{attribute 'monitoring' := 'call'}
PROPERTY OID : CHALET_BaseComponents.OTCID
GET
END_GET
END_PROPERTY

END_INTERFACE

// COMPONENTs/VnRegister-Access/FB_VnRegister_UDINT
{attribute 'no_explicit_call' := 'Do not call the body - Stick to OOP'}
FUNCTION_BLOCK FB_VnRegister_UDINT EXTENDS FB_VnRegister_Base
VAR
	{attribute 'hide'}
	nValue : UDINT;
	
	{attribute 'hide'}	
	fbVnReadRegister_UDINT : FB_VN_ReadRegister_UDINT;
	{attribute 'hide'}
	fbVnWriteRegister_UDINT : FB_VN_WriteRegister_UDINT;
END_VAR

METHOD FB_init : BOOL
VAR_INPUT
	bInitRetains : BOOL; // if TRUE, the retain variables are initialized (warm start / cold start)
	bInCopyCode : BOOL;  // if TRUE, the instance afterwards gets moved into the copy code (online change)
	
	ipCameraConnection : I_GigEVision_Register_Connection;
	nAddress : GVCP_REGISTER_ADDRESS;
    nEndian  : UINT;
END_VAR
VAR_INST
	{attribute 'hide'}
	bFBInitCalledOnce : BOOL; //Do the following code once during start up and not during onlinechange
END_VAR
//Do the following code once during start up and not during onlinechange
IF NOT bFBInitCalledOnce THEN 
	nCtsVnRegisterObject := nCtsVnRegisterObject +1;
	

	THIS^.nEndian 		:= nEndian;
	
	//Copy ObjectId from Camera to this fbVnReadRegister.
	MEMCPY(destAddr := ADR(fbVnReadRegister_UDINT.oidITcVnGevImageProvider), srcAddr:=ADR(SUPER^.OidCamera), n:= SIZEOF(SUPER^.OidCamera));
	MEMCPY(destAddr := ADR(fbVnWriteRegister_UDINT.oidITcVnGevImageProvider), srcAddr:=ADR(SUPER^.OidCamera), n:= SIZEOF(SUPER^.OidCamera));

	//Force to do an init after set OID
	fbVnReadRegister_UDINT.FB_init(FALSE,FALSE);	
	fbVnWriteRegister_UDINT.FB_init(FALSE,FALSE);
END_IF

bFBInitCalledOnce := TRUE;
END_METHOD

METHOD Update : HRESULT
SUPER^.Update();


fbVnReadRegister_UDINT(
	nAddress:= SUPER^.nAddress, 
	nEndian:= SUPER^.nEndian, 
	bRead:= SUPER^.bExecuteRead, 
	bBusy=> SUPER^.bReadBusy, 
	bError=> SUPER^.bReadError
	);
IF fbRTrigReadDone.Q AND THIS^.bWriteDone THEN
	nValue := fbVnReadRegister_UDINT.nValue;
END_IF
	
	
fbVnWriteRegister_UDINT(
	nAddress:= SUPER^.nAddress, 
	nValue:= nValue,  
	nEndian:= SUPER^.nEndian,   
	bWrite:= SUPER^.bExecuteWrite, 
	bBusy=> SUPER^.bWriteBusy, 
	bError=> SUPER^.bWriteError,
	);
END_METHOD

{attribute 'monitoring':='call'}
PROPERTY Value : UDINT
GET
Value := nValue;
END_GET
SET
nValue := Value;

//Trigger a new write cycle
THIS^.bWriteDone 	:= FALSE;
END_SET
END_PROPERTY

END_FUNCTION_BLOCK

// COMPONENTs/VnRegister-Access/internal/FB_VnRegister_Base
(* This FB is abstract and is the base class  *)
FUNCTION_BLOCK ABSTRACT FB_VnRegister_Base EXTENDS FB_CH_Object IMPLEMENTS I_VnRegister_Status
VAR

	{attribute 'hide'}
	bErrorInvalideInterface : BOOL;
	
	{attribute 'hide'}	
	OidCamera : OTCID;
	{attribute 'hide'}
	//The address of the first byte to write to the camera 
    nAddress : GVCP_REGISTER_ADDRESS;
	{attribute 'hide'}
	//The endianness of the register. 0 = Big, 1 = Little. Default: 0
    nEndian  : UINT;
	
	//in the event of a connection interruption to the device, either a read under write command is repeated
	{attribute 'hide'}
	eCommandToRepeadAfterReconnect : (READ, WRITE) := READ;
	
	//Read/write 
	{attribute 'hide'}
	bReadDone : BOOL;
	{attribute 'hide'}
	fbRTrigReadDone : R_TRIG();
	{attribute 'hide'}
	nSeqRead : UINT;
	{attribute 'hide'}
	bExecuteRead : BOOL;
	{attribute 'hide'}
	bReadError : BOOL;
	{attribute 'hide'}
	bReadBusy : BOOL;
	
	{attribute 'hide'}
	bWriteDone : BOOL := TRUE;
	{attribute 'hide'}
	nSeqWrite : UINT;

	{attribute 'hide'}
	bExecuteWrite : BOOL;	
	{attribute 'hide'}
	bWriteError : BOOL;
	{attribute 'hide'}
	bWriteBusy : BOOL;
	
	{attribute 'hide'}
	fbDelayOnError : TON := ( PT:= T#100MS);
END_VAR
VAR_STAT
	{attribute 'hide'}
	nCtsVnRegisterObject : UDINT;
	{attribute 'hide'}
	nCtsReadActive : UDINT;
	{attribute 'hide'}
	nCtsWriteActive : UDINT;
END_VAR

{attribute 'monitoring':='call'}
PROPERTY Error : BOOL
GET
Error := THIS^.bReadError OR THIS^.bWriteError OR THIS^.bErrorInvalideInterface;
END_GET
END_PROPERTY

METHOD FB_init : BOOL
VAR_INPUT
	bInitRetains : BOOL; // if TRUE, the retain variables are initialized (warm start / cold start)
	bInCopyCode : BOOL;  // if TRUE, the instance afterwards gets moved into the copy code (online change)
	
	ipCameraConnection : I_GigEVision_Register_Connection;
    nAddress : GVCP_REGISTER_ADDRESS;
END_VAR

VAR_INST
	{attribute 'hide'}
	bFBInitCalledOnce : BOOL; //Do the following code once during start up and not during onlinechange
END_VAR
//Do the following code once during start up and not during onlinechange
IF NOT bFBInitCalledOnce THEN 
	THIS^.nAddress 		:= nAddress;

	IF ipCameraConnection <> 0 THEN
		OidCamera := ipCameraConnection.OID;
	ELSE
		bErrorInvalideInterface := TRUE;
	END_IF
END_IF

bFBInitCalledOnce := TRUE;
END_METHOD

METHOD Initialize : HRESULT
IF eCommandToRepeadAfterReconnect = READ THEN
	//the reading of the parameter should be restarted again
	THIS^.bReadDone := FALSE;
END_IF

IF eCommandToRepeadAfterReconnect = WRITE THEN
	//the reading of the parameter should be restarted again
	THIS^.bWriteDone := FALSE;
END_IF


Initialize := S_OK;
END_METHOD

{attribute 'monitoring':='call'}
PROPERTY OID : OTCID
GET
OID := OidCamera;
END_GET
END_PROPERTY

{attribute 'monitoring':='call'}
PROPERTY ReadDone : BOOL
GET
ReadDone := bReadDone;
END_GET
SET
//Only allow set to FALSE
IF NOT ReadDone THEN
	bReadDone := FALSE;
END_IF
END_SET
END_PROPERTY

METHOD Update : HRESULT
IF bErrorInvalideInterface THEN
	//Error
	RETURN;
END_IF


(*--- Read ---*)
bExecuteRead := FALSE;
CASE nSeqRead OF
	0: //Start/Restart if required
		IF NOT bReadDone  AND bWriteDone(* Write has higher priority*) AND (nCtsReadActive < VisionParameterlist.MAX_VN_REGISTER_READ) AND (nSeqWrite = 0) THEN
			bExecuteRead := TRUE; // Rising edge	
			nCtsReadActive := nCtsReadActive +1;	
			nSeqRead := 1;
		END_IF
	
	1: //Check if done or error
		IF bReadError THEN
			//Error
			nSeqRead := 99;
			fbDelayOnError.IN := TRUE;
			nCtsReadActive := nCtsReadActive -1;	
			
		ELSIF NOT bReadBusy AND NOT bReadError THEN
			//Done
			THIS^.bReadDone := TRUE;
			nSeqRead := 0;
			nCtsReadActive := nCtsReadActive -1;	
			
		ELSE
			;//Busy
		END_IF	
		
	99: // Delay on error to reduce amount of errors
		IF fbDelayOnError.Q THEN
			fbDelayOnError.IN := FALSE;
			nSeqRead := 0;
		END_IF
END_CASE

fbRTrigReadDone(CLK := THIS^.bReadDone);




(*--- Write ---*)
bExecuteWrite := FALSE;
CASE nSeqWrite OF
	0: //Start/Restart if required
		IF NOT bWriteDone AND (nCtsWriteActive < VisionParameterlist.MAX_VN_REGISTER_WRITE) AND (nSeqRead = 0) THEN
			bExecuteWrite := TRUE; // Rising edge	
			nCtsWriteActive := nCtsWriteActive +1;	
			nSeqWrite := 1;
		END_IF
	
	1: //Check if done or error
		IF bWriteError THEN
			//Error
			nSeqWrite := 99;
			fbDelayOnError.IN := TRUE;
			nCtsWriteActive := nCtsWriteActive -1;	
			
		ELSIF NOT bWriteBusy AND NOT bWriteError THEN
			//Done
			THIS^.bWriteDone := TRUE;
			nSeqWrite := 0;
			nCtsWriteActive := nCtsWriteActive -1;
			
		ELSE
			;//Busy
		END_IF	
		
	99: // Delay on error to reduce amount of errors
		IF fbDelayOnError.Q THEN
			fbDelayOnError.IN := FALSE;
			nSeqWrite := 0;
		END_IF		

END_CASE



//Update
fbDelayOnError();
END_METHOD

{attribute 'monitoring':='call'}
PROPERTY WriteDone : BOOL
GET
WriteDone := bWriteDone;
END_GET
SET
//Only allow set to FALSE
IF NOT WriteDone THEN
	bWriteDone := FALSE;
END_IF

//in the event of a connection interruption to the device, either a read under write command is repeated
eCommandToRepeadAfterReconnect := WRITE;
END_SET
END_PROPERTY

END_FUNCTION_BLOCK

// COMPONENTs/VnRegister-Access/internal/I_VnRegister_Status
INTERFACE I_VnRegister_Status

{attribute 'monitoring':='call'}
PROPERTY ReadDone : BOOL
GET
END_GET
END_PROPERTY

{attribute 'monitoring':='call'}
PROPERTY WriteDone : BOOL
GET
END_GET
END_PROPERTY

END_INTERFACE

// COMPONENTs/VnRegister-Access/FB_VnRegister_Memory
{attribute 'no_explicit_call' := 'Do not call the body - Stick to OOP'}
FUNCTION_BLOCK FB_VnRegister_Memory EXTENDS FB_VnRegister_Base
VAR
	{attribute 'hide'}
	ValueBuffer 			: ARRAY[0..535] OF BYTE;
	nLength       : UINT;
	
	{attribute 'hide'}	
	fbVnReadRegister_Memory	: FB_VN_ReadMemory;
	{attribute 'hide'}
	fbVnWriteRegister_Memory : FB_VN_WriteMemory;
END_VAR

METHOD FB_init : BOOL
VAR_INPUT
	bInitRetains : BOOL; // if TRUE, the retain variables are initialized (warm start / cold start)
	bInCopyCode : BOOL;  // if TRUE, the instance afterwards gets moved into the copy code (online change)
	
	ipCameraConnection : I_GigEVision_Register_Connection;
	nAddress : GVCP_REGISTER_ADDRESS;
	//The number of bytes to write, starting at nAddress (must be a multiple of 4, not more than 536)
	nLength       : UINT; 
END_VAR
VAR_INST
	{attribute 'hide'}
	bFBInitCalledOnce : BOOL; //Do the following code once during start up and not during onlinechange
END_VAR
//Do the following code once during start up and not during onlinechange
IF NOT bFBInitCalledOnce THEN 
	nCtsVnRegisterObject := nCtsVnRegisterObject +1;
	

	THIS^.nLength 		:=  LIMIT(4, nLength, 536);
	
	//Copy ObjectId from Camera to this fbVnReadRegister.
	MEMCPY(destAddr := ADR(fbVnReadRegister_Memory.oidITcVnGevImageProvider), srcAddr:=ADR(SUPER^.OidCamera), n:= SIZEOF(SUPER^.OidCamera));
	MEMCPY(destAddr := ADR(fbVnWriteRegister_Memory.oidITcVnGevImageProvider), srcAddr:=ADR(SUPER^.OidCamera), n:= SIZEOF(SUPER^.OidCamera));

	//Force to do an init after set OID
	fbVnReadRegister_Memory.FB_init(FALSE,FALSE);	
	fbVnWriteRegister_Memory.FB_init(FALSE,FALSE);
END_IF

bFBInitCalledOnce := TRUE;
END_METHOD

METHOD ReadData : BOOL
VAR_INPUT
	//ADR(destination)
	pBuffer  : PVOID; 
END_VAR
MEMCPY(destAddr := pBuffer, srcAddr:=ADR(ValueBuffer), n:= nLength);
END_METHOD

METHOD Update : HRESULT
SUPER^.Update();

fbVnReadRegister_Memory(
	nAddress:= SUPER^.nAddress, 
	nLength:= nLength, 
	pBuffer:= ADR(ValueBuffer), 
	bRead:= SUPER^.bExecuteRead, 
	bBusy=> SUPER^.bReadBusy, 
	bError=> SUPER^.bReadError
	);
	
fbVnWriteRegister_Memory(
	nAddress:= SUPER^.nAddress, 
	nLength:= nLength, 
	pData:= ADR(ValueBuffer), 
	bWrite:= SUPER^.bExecuteWrite, 
	bBusy=> SUPER^.bWriteBusy, 
	bError=> SUPER^.bWriteError,
	);
END_METHOD

METHOD WriteData : BOOL
VAR_INPUT
	//ADR(source)
	pBuffer  : PVOID; 
END_VAR
MEMCPY(destAddr := ADR(ValueBuffer), srcAddr:= pBuffer, n:= nLength);

//Trigger a new write cycle
THIS^.bWriteDone 	:= FALSE;
END_METHOD

END_FUNCTION_BLOCK

// COMPONENTs/ImageProvider/Camera/FB_GigE_Vision
{attribute 'no_explicit_call' := 'Do not call the body - Stick to OOP'}
FUNCTION_BLOCK FB_GigE_Vision EXTENDS FB_ImageProvider_Base IMPLEMENTS I_GigEVision_Mode, I_GigEVision_Register_Connection
VAR
	fbCamera 						: FB_VN_GevCameraControl;	// Interface object for camera use
	
	{attribute 'hide'}
	fbCameraWriteExposureTime		: FB_VN_WriteRegister_UDINT;// Interface object for camera configuration
	{attribute 'hide'}
	bResetCommand	: BOOL;
END_VAR

{attribute 'monitoring' := 'call'}
PROPERTY Exposure_1us : UDINT
GET
Exposure_1us := THIS^.fbCameraWriteExposureTime.nValue;
END_GET
SET
THIS^.fbCameraWriteExposureTime.nValue := Exposure_1us;
THIS^.fbCamera.StopAcquisition();
END_SET
END_PROPERTY

METHOD FB_init : BOOL
VAR_INPUT
	bInitRetains : BOOL; // if TRUE, the retain variables are initialized (warm start / cold start)
	bInCopyCode : BOOL;  // if TRUE, the instance afterwards gets moved into the copy code (online change)
	
	(*The register address identifies the camera register to be addressed. 
		It is of the type GVCP_REGISTER_ADDRESS, which is an alias of the type UDINT. Thus, all register addresses have a size of 4 bytes. 
		The register address of a camera parameter can be seen at the respective point in the configuration tree of the GigE Vision camera instance*)
	nAddressExposureTime : GVCP_REGISTER_ADDRESS;
	
	
	(*Endianess describes the order in which the bytes of a camera register are arranged. 
		This does not need to be considered any further in terms of the application and can be adopted as a property of the respective parameter of the configuration tree of the GigE Vision camera instance.
		A Big Endian is represented by nEndian := 0 and a Small Endian by nEndian := 1. Big Endian is the default.*)
	nEndian : UINT; 
END_VAR
VAR_INST
	{attribute 'hide'}
	bFBInitCalledOnce : BOOL; //Do the following code once during start up and not during onlinechange
END_VAR
//Do the following code once during start up and not during onlinechange
IF NOT bFBInitCalledOnce THEN 
	
	THIS^.fbCameraWriteExposureTime.nAddress := nAddressExposureTime;
	THIS^.fbCameraWriteExposureTime.nEndian := nEndian;
	THIS^.fbCameraWriteExposureTime.nTimeout := T#500MS;
	THIS^.fbCameraWriteExposureTime.nValue	:= 10000;
	
//Copy OID from camera instead of symbol initialization
MEMCPY(destAddr := ADR(fbCameraWriteExposureTime.oidITcVnGevImageProvider), srcAddr:=ADR(THIS^.fbCamera.oidITcVnGevImageProvider), n:= SIZEOF(fbCameraWriteExposureTime.oidITcVnGevImageProvider));

END_IF

bFBInitCalledOnce := TRUE;
END_METHOD

//Reference to base function block
PROPERTY GevCameraControl : REFERENCE TO FB_VN_GevCameraControl
GET
GevCameraControl REF= THIS^.fbCamera;
END_GET
END_PROPERTY

METHOD Initialize : HRESULT
VAR 
	fbTaskInfo		 : PlcTaskSystemInfo;
END_VAR
VAR_INST
	//This error cannot be reset. Requires a reset cold
	{attribute 'hide'}	
	fbInitError : FB_TcAlarm;
END_VAR
SUPER^.Initialize();


// Object id of ImagePoovider is not set
IF THIS^.fbCamera.oidITcVnGevImageProvider = 0 THEN
	IF NOT fbInitError.bRaised THEN 
		//This error cannot be reset. Requires a reset cold
		fbInitError.CreateEx(stEventEntry:=TC_EVENTS.CHALET_Vision_Events.ObjectIdNotSet, ipSourceInfo := THIS^.fbSourceInfo, bWithConfirmation := FALSE);
		fbInitError.Raise(0);
	END_IF
	Initialize := E_FAIL;
	RETURN;
END_IF

// Object id of ImagePoovider is not set
IF THIS^.fbCameraWriteExposureTime.oidITcVnGevImageProvider = 0 THEN
	IF NOT fbInitError.bRaised THEN 
		//This error cannot be reset. Requires a reset cold
		fbInitError.CreateEx(stEventEntry:=TC_EVENTS.CHALET_Vision_Events.ObjectIdNotSet, ipSourceInfo := THIS^.fbSourceInfo, bWithConfirmation := FALSE);
		fbInitError.Raise(0);
	END_IF
	Initialize := E_FAIL;
	RETURN;
END_IF
END_METHOD

{attribute 'monitoring' := 'call'}
PROPERTY OID : CHALET_BaseComponents.OTCID
GET
OID := THIS^.fbCamera.oidITcVnGevImageProvider;
END_GET
END_PROPERTY

METHOD Reset : HRESULT
VAR_INPUT
END_VAR
bResetCommand := TRUE;
END_METHOD

METHOD PUBLIC Softtrigger : HRESULT
(* Check if not in wrong state *)
IF NOT ((THIS^.eState = ETcVnCameraState.TCVN_CS_ACQUIRING) OR (THIS^.eState = ETcVnCameraState.TCVN_CS_OPENED)) THEN
	Softtrigger := E_FAIL;
	RETURN;
END_IF


THIS^.eState := ETcVnCameraState.TCVN_CS_TRIGGERING;

// Trigger image
Softtrigger := fbCamera.TriggerImage();
END_METHOD

{attribute 'monitoring' := 'call'}
PROPERTY State : ETcVnCameraState
GET
State := THIS^.eState;
END_GET
END_PROPERTY

METHOD TryGetImage : HRESULT
VAR_INPUT
	stImageWithInfo : REFERENCE TO ST_ImageWithInfo;
END_VAR
IF NOT __ISVALIDREF(stImageWithInfo) THEN
	//Error, invalide input
	TryGetImage := E_FAIL;
	RETURN;
END_IF


(* Release the old image before overwriting it with the new one *)	
IF stImageWithInfo.ipImage <> 0 THEN
	FW_SafeRelease(ADR(stImageWithInfo.ipImage));
END_IF

(*  Lock the image to prevent multiple access *)
(*	🔒 LOCKED FROM HERE --------------------------------------------- *)
IF THIS^.fbCrititcalSection.Enter() THEN
	
	(* Get current image from camera *)
	TryGetImage := fbCamera.GetCurrentImageWithGvspInfo(
						ipImage := stImageWithInfo.ipImage,
						stGvspInfo := stImageWithInfo.stGvspInfo
						);

	(* Get image info from received image *)
	F_VN_GetImageInfo(	ipImage:=stImageWithInfo.ipImage, 
						stImageInfo:=stImageWithInfo.stInfo, 
						hrPrev:=TryGetImage );
	
	(* for a camera a fictitious name *)
	stImageWithInfo.sCurrentImageFileName := TO_STRING(stImageWithInfo.stGvspInfo.BlockId);			

	(*	🔓 LOCKED TO HERE ----------------------------------------------- *)
	THIS^.fbCrititcalSection.Leave();
END_IF
END_METHOD

METHOD Update : HRESULT
(* Get current source state *)					
eState := fbCamera.GetState();

(* Source state machine *)
CASE eState OF
	TCVN_CS_INITIAL, TCVN_CS_INITIALIZING:
		fbCameraWriteExposureTime.bWrite := FALSE;	
		fbFeedback.ActiveCommand := 'InitializeCamera';
		fbFeedback.hr := fbCamera.InitializeCamera();

	TCVN_CS_INITIALIZED,  TCVN_CS_OPENING:
		fbCameraWriteExposureTime.bWrite := FALSE;	
		fbFeedback.ActiveCommand := 'OpenCamera';
		fbFeedback.hr := fbCamera.OpenCamera();
		
	TCVN_CS_OPENED:
		(* Write camera Parameters*)
		IF (fbCameraWriteExposureTime.bWrite AND NOT fbCameraWriteExposureTime.bBusy AND NOT fbCameraWriteExposureTime.bError) THEN
			(* Done - Process with state machine *)
			fbFeedback.ActiveCommand := 'StartAcquisition';
			fbFeedback.hr := fbCamera.StartAcquisition();
			fbCameraWriteExposureTime.bWrite := FALSE;
		ELSIF NOT fbCameraWriteExposureTime.bWrite THEN
			(* Not startet - Start now *)
			fbFeedback.ActiveCommand := 'WriteExposureTime';
			fbFeedback.Busy := TRUE;
			fbCameraWriteExposureTime.bWrite := TRUE;
		ELSIF fbCameraWriteExposureTime.bError THEN
			(* Error - Toggle writte signal *)
			fbCameraWriteExposureTime.bWrite := FALSE;
		END_IF
		
	TCVN_CS_STARTACQUISITION:
		fbFeedback.ActiveCommand := 'StartAcquisition';
		fbFeedback.hr := fbCamera.StartAcquisition();
		
		
	TCVN_CS_STOPACQUISITION:
		fbFeedback.ActiveCommand := 'StopAcquisition';
		fbFeedback.hr := fbCamera.StopAcquisition();
		
	TCVN_CS_ACQUIRING:
	;


		
	TCVN_CS_TRIGGERING:
		fbFeedback.ActiveCommand := 'TriggerImage';
		fbFeedback.hr := fbCamera.TriggerImage();
		
	TCVN_CS_ERROR:	
		//(* Raise Alarm *)
		//IF NOT THIS^.fbAlarmGeneral.bRaised THEN	
		//	THIS^.stAlarmCode.sErrCode := DWORD_TO_HEXSTR(TO_DWORD(THIS^.hrSource), 0, FALSE);;
		//	THIS^.stAlarmCode.sAdsCode := RIGHT(THIS^.stAlarmCode.sErrCode,3);
		//	THIS^.fbAlarmGeneral.ipArguments.Clear();
		//	THIS^.fbAlarmGeneral.ipArguments.AddString(stAlarmCode.sErrCode);
		//	THIS^.fbAlarmGeneral.ipArguments.AddString(stAlarmCode.sAdsCode);
		//	THIS^.fbAlarmGeneral.Raise(0);	
		//END_IF
		
		(* Reset if commanded *)
		IF 	THIS^.bResetCommand THEN
			fbFeedback.ActiveCommand := 'Reset';
			fbFeedback.hr := THIS^.fbCamera.Reset();			
		END_IF
END_CASE

(* Clear Alarm if not in Error-State *)
IF eState <> TCVN_CS_ERROR THEN
	THIS^.bResetCommand := FALSE;
END_IF


(* Update camera parameters*)
fbCameraWriteExposureTime();
END_METHOD

END_FUNCTION_BLOCK

// COMPONENTs/ImageProvider/ImageFromFile/FB_ImageFromFile
{attribute 'no_explicit_call' := 'Do not call the body - Stick to OOP'}
FUNCTION_BLOCK FB_ImageFromFile EXTENDS FB_ImageProvider_Base IMPLEMENTS I_ImageFromFile_Mode
VAR
	fbFileSourceCtl 	: FB_VN_FileSourceControl;	// Interface object for file source use
	{attribute 'hide'}
	sRequestSpecificImageName : STRING;
	{attribute 'hide'}
	nTimeNextTrigger  	: T_DCTIME64; 
	{attribute 'hide'}
	bResetCommand	: BOOL;
	{attribute 'hide'}
	sLastImageFileName : STRING(500);
END_VAR

//Reference to base function block
PROPERTY FileSourceControl : REFERENCE TO FB_VN_FileSourceControl
GET
FileSourceControl REF= THIS^.fbFileSourceCtl;
END_GET
END_PROPERTY

METHOD Initialize : HRESULT
VAR

END_VAR
VAR_INST
	//This error cannot be reset. Requires a reset cold
	{attribute 'hide'}	
	fbInitError : FB_TcAlarm;
END_VAR
SUPER^.Initialize();

// Object id of ImagePoovider is not set
IF THIS^.fbFileSourceCtl.oidITcVnFileImageProvider = 0 THEN
	IF NOT fbInitError.bRaised THEN 
		//This error cannot be reset. Requires a reset cold
		fbInitError.CreateEx(stEventEntry:=TC_EVENTS.CHALET_Vision_Events.ObjectIdNotSet, ipSourceInfo := THIS^.fbSourceInfo, bWithConfirmation := FALSE);
		fbInitError.Raise(0);
	END_IF
	Initialize := E_FAIL;
	RETURN;
END_IF
END_METHOD

PROPERTY LastImageFileName : STRING(500)
GET
LastImageFileName := sLastImageFileName;
END_GET
END_PROPERTY

{attribute 'monitoring' := 'call'}
PROPERTY OID : CHALET_BaseComponents.OTCID
GET
OID := THIS^.fbFileSourceCtl.oidITcVnFileImageProvider;
END_GET
END_PROPERTY

{attribute 'monitoring' := 'call'}
//Next trigger will load a specific image in the list by name. ('' = any image)
PROPERTY RequestSpecificImageName : STRING
GET
RequestSpecificImageName := sRequestSpecificImageName;
END_GET
SET
sRequestSpecificImageName := RequestSpecificImageName;
END_SET
END_PROPERTY

METHOD Reset : HRESULT
VAR_INPUT
END_VAR
bResetCommand := TRUE;
END_METHOD

{attribute 'monitoring' := 'call'}
PROPERTY State : ETcVnCameraState
GET
State := THIS^.eState;
END_GET
END_PROPERTY

METHOD Trigger : HRESULT
VAR_INPUT
	nTimeStamp : T_DCTIME64;
END_VAR
IF THIS^.Operational AND NOT THIS^.fbFeedback.Busy THEN	
	
	//Stor the requestet time internal
	THIS^.nTimeNextTrigger := nTimeStamp;
	
	Trigger := S_OK;
ELSE
	Trigger := E_FAIL;
END_IF
END_METHOD

METHOD TryGetImage : HRESULT
VAR_INPUT
	stImageWithInfo : REFERENCE TO ST_ImageWithInfo;
END_VAR
IF NOT __ISVALIDREF(stImageWithInfo) THEN
	//Error, invalide input
	TryGetImage := E_FAIL;
	RETURN;
END_IF


(* Release the old image before overwriting it with the new one *)	
IF stImageWithInfo.ipImage <> 0 THEN
	FW_SafeRelease(ADR(stImageWithInfo.ipImage));
END_IF

(*  Lock the image to prevent multiple access *)
(*	🔒 LOCKED FROM HERE --------------------------------------------- *)
IF THIS^.fbCrititcalSection.Enter() THEN
	
	(* Get current image from camera *)
	TryGetImage := fbFileSourceCtl.GetCurrentImageAndFileName(	ipImage := stImageWithInfo.ipImage, 
																sFileName := sLastImageFileName, 
																nMaxLen := SIZEOF(sLastImageFileName)/SIZEOF(STRING(1))
																);

	(* Get image info from received image *)
	F_VN_GetImageInfo(	ipImage:=stImageWithInfo.ipImage, 
						stImageInfo:=stImageWithInfo.stInfo, 
						hrPrev:=TryGetImage );
	
	(* Not used for image from file *)					
	//stImageWithInfo.stGvspInfo

	(* Store file name *)
	stImageWithInfo.sCurrentImageFileName := sLastImageFileName;			
						
	(*	🔓 LOCKED TO HERE ----------------------------------------------- *)
	THIS^.fbCrititcalSection.Leave();
END_IF
END_METHOD

METHOD Update : HRESULT
(* Get current source state *)					
eState := fbFileSourceCtl.GetState();

(* Source state machine *)
CASE eState OF
	TCVN_CS_INITIAL, TCVN_CS_INITIALIZING, TCVN_CS_INITIALIZED, TCVN_CS_OPENING, TCVN_CS_STARTACQUISITION, TCVN_CS_OPENED:	
		fbFeedback.ActiveCommand := 'StartAcquisition';
		fbFeedback.hr := fbFileSourceCtl.StartAcquisition();

	TCVN_CS_STOPACQUISITION:
		fbFeedback.ActiveCommand := 'StopAcquisition';
		fbFeedback.hr := fbFileSourceCtl.StopAcquisition();
		
	TCVN_CS_ACQUIRING:
		fbFeedback.ActiveCommand := 'TriggerImage';
		IF (THIS^.nTimeNextTrigger = 0) THEN
			fbFeedback.Done := TRUE; //wait for a trigger
			
		ELSIF (F_GetCurDcTaskTime64()  >=  THIS^.nTimeNextTrigger)  THEN
			//Clear
			THIS^.nTimeNextTrigger := 0;
			
			IF sRequestSpecificImageName <> '' THEN
				//Trigger image by name
				fbFeedback.hr := fbFileSourceCtl.TriggerImageByName(sRequestSpecificImageName);
			ELSE
				//Any image
				fbFeedback.hr := fbFileSourceCtl.TriggerImage();
			END_IF
			
		ELSIF (THIS^.nTimeNextTrigger <> 0) THEN
			fbFeedback.Busy := TRUE; //wait until trigger moment starts
		END_IF

		
	TCVN_CS_TRIGGERING:
		fbFeedback.ActiveCommand := 'TriggerImage';
		fbFeedback.hr := fbFileSourceCtl.TriggerImage();
		
	TCVN_CS_ERROR:
		(* Reset if commanded *)
		IF THIS^.bResetCommand THEN
			fbFeedback.ActiveCommand := 'Reset';
			fbFeedback.hr := THIS^.fbFileSourceCtl.Reset();			
		END_IF		
END_CASE

(* Clear Alarm if not in Error-State *)
IF eState <> TCVN_CS_ERROR THEN
	THIS^.bResetCommand := FALSE;
END_IF

Update := S_OK;
END_METHOD

END_FUNCTION_BLOCK

// COMPONENTs/ImageProvider/ImageFromFile/I_ImageFromFile_Mode
INTERFACE I_ImageFromFile_Mode

{attribute 'monitoring' := 'call'}
//Next trigger will load a specific image in the list by name. ('' = any image)
PROPERTY RequestSpecificImageName : STRING
GET
END_GET
SET
END_SET
END_PROPERTY

METHOD Trigger : HRESULT
VAR_INPUT
	nTimeStamp : T_DCTIME64;
END_VAR
END_METHOD

END_INTERFACE

// COMPONENTs/Mode/Combined illumination and camera triggers/FB_VisionMode_Pulse_combined
{attribute 'no_explicit_call' := '[FB_VisionMode_Pulse] Do not call the body - Stick to OOP'}
//Pulse - A trigger activates an image acquisition with simultaneous triggering of the lighting 
FUNCTION_BLOCK FB_VisionMode_Pulse_combined EXTENDS FB_VisionMode_Base IMPLEMENTS I_VisionMode_Pulse_combined
VAR
	{attribute 'hide'}
	bInitDone : BOOL;
	{attribute 'hide'}
	nLastTriggerTime : T_DCTIME64;
	
	(* Supported/requested interfaces. Minimum one must be supported per ImageProvider/CameraController/IlluminationController *)
	(* ImageProvider *)
	ipGigeVision_Mode 	: I_GigEVision_Mode;	
	ipImageFromFile_Mode	: I_ImageFromFile_Mode;	
	
	(* Supported/requested interfaces. Minimum one must be supported per ImageProvider/CameraController/IlluminationController *)
	(* CameraController *)
	ipHwTimestamp_Mode 		: I_HwTimestamp_Mode;
	ipSwTimestamp_Mode		: I_SwTimestamp_Mode;
	ipGigeSoftwaretrigger 	: I_GigeSoftTrigger_Mode;
	
	(* Supported/requested interfaces. Minimum one must be supported per ImageProvider/CameraController/IlluminationController *)
	(* lluminationController 1 *)
	ipVIx2000_Mode_1 		: I_VIx2000_Mode;
	ipSingleOutput_Mode_1 	: I_IlluminationSingleOutput_Mode;
		
	(* Supported/requested interfaces. Minimum one must be supported per ImageProvider/CameraController/IlluminationController *)
	(* lluminationController 2 *)
	ipVIx2000_Mode_2 	: I_VIx2000_Mode;
	ipSingleOutput_Mode_2 	: I_IlluminationSingleOutput_Mode;
	
END_VAR

METHOD Configure : HRESULT
VAR_INPUT
	nOrange 	: UINT(0..511); //0-511
	nGreen 		: UINT(0..511); //0-511
	nBlue 		: UINT(0..511); //0-511
	nInfrared 	: UINT(0..511); //0-511
//	nExposureDelay_100ns : UDINT;	//Camera start at triggertime, illumination starts this time earlier
	nExposure_1us : UDINT;			//Camera 
	nIlluminationDuration_1us: UDINT;
	nIlluminationOverride : USINT(1..100); // 1-100
END_VAR
VAR
	hr : HRESULT;
END_VAR
IF NOT bInitDone THEN
	Configure := E_FAIL;
	RETURN;
END_IF	


(* CameraController *)
(* Decide here how the hardware is to be controlled based on the interface that was found *)
IF ipHwTimestamp_Mode <> 0 THEN
//	ipHwTimestamp_Mode.TriggerDelay_1ns := nExposureDelay_100ns; zzz clean up
	ipHwTimestamp_Mode.Duration_1us := nExposure_1us;// + TO_UDINT(nExposureDelay_100ns/10); //exposure + warm up time
END_IF

IF ipSwTimestamp_Mode <> 0 THEN
//	ipSwTimestamp_Mode.TriggerDelay_1ns := nExposureDelay_100ns;
END_IF

IF ipGigeSoftwaretrigger <> 0 THEN
	ipGigeSoftwaretrigger.GigeCamera := ipGigeVision_Mode;
//	ipGigeSoftwaretrigger.TriggerDelay_1ns := nExposureDelay_100ns;
END_IF
 


(* ImageProvider *)
(* Decide here how the hardware is to be controlled based on the interface that was found *)
IF ipGigeVision_Mode <> 0 THEN
	ipGigeVision_Mode.Exposure_1us := nExposure_1us;
END_IF




(* lluminationController1 *)
(* Decide here how the hardware is to be controlled based on the interface that was found *)
IF ipVIx2000_Mode_1 <> 0 THEN
	hr := GetMostSignificant(hr, ipVIx2000_Mode_1.Configure(
															nOrange		:= (nOrange*nIlluminationOverride/100), 
															nGreen		:= (nGreen*nIlluminationOverride/100), 
															nBlue		:= (nBlue*nIlluminationOverride/100), 
															nInfrared	:= (nInfrared*nIlluminationOverride/100), 
															nDuration_1us:= nIlluminationDuration_1us));
END_IF




(* lluminationController2 *)
(* Decide here how the hardware is to be controlled based on the interface that was found *)
IF ipVIx2000_Mode_2 <> 0 THEN
	hr := GetMostSignificant(hr, ipVIx2000_Mode_2.Configure(
															nOrange		:= (nOrange*nIlluminationOverride/100), 
															nGreen		:= (nGreen*nIlluminationOverride/100), 
															nBlue		:= (nBlue*nIlluminationOverride/100), 
															nInfrared	:= (nInfrared*nIlluminationOverride/100), 
															nDuration_1us:= nIlluminationDuration_1us));
END_IF



Configure := hr;
END_METHOD

METHOD Initialize : HRESULT
VAR 
	bSupportedCameraController, bSupportedlluminationController1, bSupportedlluminationController2, bSupportedlImageProvider : BOOL;
END_VAR
(* CameraController *)
bSupportedCameraController := 	ToHwTimestamp_Mode(ipCameraTriggerController, ipHwTimestamp_Mode)
							OR 	ToSwTimestamp_Mode(ipCameraTriggerController, ipSwTimestamp_Mode)
							OR 	(ToImageFromFile_Mode(ipImageProvider, ipImageFromFile_Mode) AND ipCameraTriggerController=0)	//No Cameracontrolle is allowed if ImageFromFile	
							OR (ToGigeSoftTrigger_Mode(ipCameraTriggerController, ipGigeSoftwaretrigger) AND ToGigEVision_Mode(ipImageProvider, ipGigeVision_Mode));//GigE Softtrigger requires a GigE ImageProvider
							// OR ...

							
(* ImageProvider *)
bSupportedlImageProvider := ToGigEVision_Mode(ipImageProvider, ipGigeVision_Mode)	
						 OR ToImageFromFile_Mode(ipImageProvider, ipImageFromFile_Mode); 
							// OR ...

							
(* lluminationController1 *)
bSupportedlluminationController1 := 	ToVIx2000_Mode(ipIlluminationController1, ipVIx2000_Mode_1)
									OR 	ToIlluminationSingleOutput_Mode(ipIlluminationController1, ipSingleOutput_Mode_1)
									OR 	(ipIlluminationController1 = 0); //Ilumination1+2 is optional -> Empty or valide
									// OR ...

									
(* lluminationController2 *)
bSupportedlluminationController2 := 	ToVIx2000_Mode(ipIlluminationController2, ipVIx2000_Mode_2)
									OR 	ToIlluminationSingleOutput_Mode(ipIlluminationController2, ipSingleOutput_Mode_2)
									OR 	(ipIlluminationController2 = 0); //Ilumination1+2 is optional -> Empty or valide
									// OR ...

									

bInitDone := bSupportedCameraController AND bSupportedlImageProvider AND bSupportedlluminationController1 AND bSupportedlluminationController2;


IF bInitDone THEN 
	Initialize := S_OK;
ELSE
	Initialize := E_FAIL;
END_IF
END_METHOD

{attribute 'monitoring' := 'call'}
PROPERTY LastTriggerTime : T_DCTIME64
GET
LastTriggerTime := nLastTriggerTime;
END_GET
END_PROPERTY

{attribute 'monitoring' := 'call'}
// Name or description of this mode
PROPERTY Name : STRING
GET
Name := 'Acquisition with simultaneous triggering of the lighting';
END_GET
END_PROPERTY

METHOD TriggerAtDcTime : HRESULT
VAR_INPUT
	//The data type T_DCTIME64 represents the distributed clock system time (abbreviated as DC time) as a linear 64-bit integer value. 
	//The time is expressed in nanoseconds since 1/1/2000 UTC. The smallest unit is a nanosecond.
	//F_GetCurDcTickTime64()
	nDCTimeStamp	: T_DCTIME64;
END_VAR
VAR
	hr : HRESULT;
END_VAR
IF NOT bInitDone THEN
	TriggerAtDcTime := E_FAIL;
	RETURN;
END_IF	

(* Check if the trigger is minimum 3 EtherCat cycles in future *)
IF NOT (nDCTimeStamp >= THIS^.NextPossibleTriggerTime) THEN
	TriggerAtDcTime := E_FAIL;
	RETURN;
END_IF


(* CameraController *)
(* Decide here how the hardware is to be controlled based on the interface that was found *)
IF ipHwTimestamp_Mode <> 0 THEN
	hr := GetMostSignificant(hr, ipHwTimestamp_Mode.Trigger(nDCTimeStamp));
END_IF
IF ipSwTimestamp_Mode <> 0 THEN
	hr := GetMostSignificant(hr, ipSwTimestamp_Mode.Trigger(nDCTimeStamp));
END_IF
IF ipGigeSoftwaretrigger <> 0 THEN
	hr := GetMostSignificant(hr, ipGigeSoftwaretrigger.Trigger(nDCTimeStamp));
END_IF



(* ImageProvider *)
IF ipImageFromFile_Mode <> 0 THEN
	hr := GetMostSignificant(hr, ipImageFromFile_Mode.Trigger(nDCTimeStamp));
END_IF



(* lluminationController1 *)
(* Decide here how the hardware is to be controlled based on the interface that was found *)
IF ipVIx2000_Mode_1 <> 0 THEN
	hr := GetMostSignificant(hr, ipVIx2000_Mode_1.Trigger(nDCTimeStamp));
END_IF
IF ipSingleOutput_Mode_1 <> 0 THEN
	hr := GetMostSignificant(hr, ipSingleOutput_Mode_1.Trigger(nDCTimeStamp));
END_IF



(* lluminationController2 *)
(* Decide here how the hardware is to be controlled based on the interface that was found *)
IF ipVIx2000_Mode_2 <> 0 THEN
	hr := GetMostSignificant(hr, ipVIx2000_Mode_2.Trigger(nDCTimeStamp));
END_IF
IF ipSingleOutput_Mode_2 <> 0 THEN
	hr := GetMostSignificant(hr, ipSingleOutput_Mode_2.Trigger(nDCTimeStamp));
END_IF

IF hr = S_OK THEN
	THIS^.nLastTriggerTime := nDCTimeStamp;
END_IF

TriggerAtDcTime := hr;
END_METHOD

METHOD TriggerNow : HRESULT
(* Trigger the vision system *)
TriggerNow := THIS^.TriggerAtDcTime(nDCTimeStamp := THIS^.NextPossibleTriggerTime);
END_METHOD

END_FUNCTION_BLOCK

// COMPONENTs/Mode/FB_VisionMode_Base
{attribute 'no_explicit_call' := 'Do not call the body - Stick to OOP'}
FUNCTION_BLOCK ABSTRACT FB_VisionMode_Base EXTENDS FB_CH_Object IMPLEMENTS I_VisionMode_Base
VAR
	{attribute 'hide'}
	ipVisionSystem 				: I_VisionSystem;
	{attribute 'hide'}
	ipCameraTriggerController 			: I_CameraTriggerController_Base;
	{attribute 'hide'}
	ipImageProvider 			: I_ImageProvider_Base;	
	{attribute 'hide'}
	ipIlluminationController1 	: I_IlluminationController_Base;
	{attribute 'hide'}
	ipIlluminationController2 	: I_IlluminationController_Base;
	{attribute 'hide'}
END_VAR

METHOD LinkComponents : HRESULT
VAR_INPUT
	ipVisionSystem		: I_VisionSystem;
	ipCameraTriggerController	: I_CameraTriggerController_Base;
	ipImageProvider 			: I_ImageProvider_Base;	
	ipIlluminationController1 : I_IlluminationController_Base;
	ipIlluminationController2 : I_IlluminationController_Base;
END_VAR
THIS^.ipVisionSystem 				:= ipVisionSystem;
THIS^.ipCameraTriggerController 	:= ipCameraTriggerController;
THIS^.ipImageProvider 				:= ipImageProvider;
THIS^.ipIlluminationController1 	:= ipIlluminationController1;
THIS^.ipIlluminationController2 	:= ipIlluminationController2;
END_METHOD

{attribute 'monitoring' := 'call'}
// Name or description of this mode
PROPERTY ABSTRACT Name : STRING
GET
END_GET
END_PROPERTY

{attribute 'monitoring' := 'call'}
PROPERTY NextPossibleTriggerTime : T_DCTIME64
GET
VAR
	tNextPossibleTriggerTime : T_DCTIME64;
END_VAR

tNextPossibleTriggerTime := F_GetCurDcTaskTime64()(*1ns*) + 1*THIS^.ipVisionSystem.TaskCycleTimeNs(*1ns*) ;



(* CameraController *)
IF ipCameraTriggerController <> 0 THEN
	tNextPossibleTriggerTime := MAX(tNextPossibleTriggerTime, ipCameraTriggerController.NextPossibleTriggerTime);
END_IF	
	


(* lluminationController1 *)
(* Decide here how the hardware is to be controlled based on the interface that was found *)
IF ipIlluminationController1 <> 0 THEN
	tNextPossibleTriggerTime := MAX(tNextPossibleTriggerTime, ipIlluminationController1.NextPossibleTriggerTime);
END_IF



(* lluminationController2 *)
(* Decide here how the hardware is to be controlled based on the interface that was found *)
IF ipIlluminationController2 <> 0 THEN
	tNextPossibleTriggerTime := MAX(tNextPossibleTriggerTime, ipIlluminationController2.NextPossibleTriggerTime);
END_IF


NextPossibleTriggerTime := tNextPossibleTriggerTime;
END_GET
END_PROPERTY

END_FUNCTION_BLOCK

// COMPONENTs/Mode/Combined illumination and camera triggers/I_VisionMode_Pulse_combined
INTERFACE I_VisionMode_Pulse_combined

METHOD Configure : HRESULT
VAR_INPUT
	nOrange 	: UINT(0..511); //0-511
	nGreen 		: UINT(0..511); //0-511
	nBlue 		: UINT(0..511); //0-511
	nInfrared 	: UINT(0..511); //0-511
//	nExposureDelay_100ns : UDINT;	//Camera start delay after illumination start zzz
	nExposure_1us : UDINT;			//Camera 
	nIlluminationDuration_1us: UDINT;
	nIlluminationOverride : USINT(1..100); // 1-100
END_VAR
END_METHOD

{attribute 'monitoring' := 'call'}
PROPERTY LastTriggerTime : T_DCTIME64
GET
END_GET
END_PROPERTY

{attribute 'monitoring' := 'call'}
PROPERTY NextPossibleTriggerTime : T_DCTIME64
GET
END_GET
END_PROPERTY

METHOD TriggerAtDcTime : HRESULT
VAR_INPUT
	//The data type T_DCTIME64 represents the distributed clock system time (abbreviated as DC time) as a linear 64-bit integer value. 
	//The time is expressed in nanoseconds since 1/1/2000 UTC. The smallest unit is a nanosecond.
	//F_GetCurDcTickTime64()
	nDCTimeStamp	: T_DCTIME64;
END_VAR
END_METHOD

METHOD TriggerNow : HRESULT
END_METHOD

END_INTERFACE

// FUNCTIONs/Casting/ToHwTimestamp_Mode
FUNCTION ToHwTimestamp_Mode : BOOL
VAR_INPUT
	ipChObject : I_CH_OBJECT;
	ipEL2596_Mode : REFERENCE TO I_HwTimestamp_Mode;
END_VAR

VAR
	ipTmp : I_HwTimestamp_Mode;
END_VAR

(* 
   1. Test if the interface exists
   2. Test if the object implements a "Object" interface 
   3. Write reference to interface in parameter
   4. Returne TRUE if succesfull
*)
IF ipChObject <> 0 AND_THEN __QUERYINTERFACE(ipChObject,ipTmp) THEN
	ipEL2596_Mode := ipTmp;
	ToHwTimestamp_Mode := TRUE;
END_IF

END_FUNCTION

// FUNCTIONs/Casting/ToSwTimestamp_Mode
FUNCTION ToSwTimestamp_Mode : BOOL
VAR_INPUT
	ipChObject : I_CH_OBJECT;
	ipSwTimestamp_Mode : REFERENCE TO I_SwTimestamp_Mode;
END_VAR

VAR
	ipTmp : I_SwTimestamp_Mode;
END_VAR

(* 
   1. Test if the interface exists
   2. Test if the object implements a "Object" interface 
   3. Write reference to interface in parameter
   4. Returne TRUE if succesfull
*)
IF ipChObject <> 0 AND_THEN __QUERYINTERFACE(ipChObject,ipTmp) THEN
	ipSwTimestamp_Mode := ipTmp;
	ToSwTimestamp_Mode := TRUE;
END_IF

END_FUNCTION

// FUNCTIONs/Casting/ToImageFromFile_Mode
FUNCTION ToImageFromFile_Mode : BOOL
VAR_INPUT
	ipChObject : I_CH_OBJECT;
	ipImageFromFile_Mode : REFERENCE TO I_ImageFromFile_Mode;
END_VAR

VAR
	ipTmp : I_ImageFromFile_Mode;
END_VAR

(* 
   1. Test if the interface exists
   2. Test if the object implements a "Object" interface 
   3. Write reference to interface in parameter
   4. Returne TRUE if succesfull
*)
IF ipChObject <> 0 AND_THEN __QUERYINTERFACE(ipChObject,ipTmp) THEN
	ipImageFromFile_Mode := ipTmp;
	ToImageFromFile_Mode := TRUE;
END_IF

END_FUNCTION

// FUNCTIONs/Casting/ToGigeSoftTrigger_Mode
FUNCTION ToGigeSoftTrigger_Mode : BOOL
VAR_INPUT
	ipChObject : I_CH_OBJECT;
	iGigeSoftTrigger_Mode : REFERENCE TO I_GigeSoftTrigger_Mode;
END_VAR

VAR
	ipTmp : I_GigeSoftTrigger_Mode;
END_VAR

(* 
   1. Test if the interface exists
   2. Test if the object implements a "Object" interface 
   3. Write reference to interface in parameter
   4. Returne TRUE if succesfull
*)
IF ipChObject <> 0 AND_THEN __QUERYINTERFACE(ipChObject,ipTmp) THEN
	iGigeSoftTrigger_Mode := ipTmp;
	ToGigeSoftTrigger_Mode := TRUE;
END_IF

END_FUNCTION

// FUNCTIONs/Casting/ToGigEVision_Mode
FUNCTION ToGigEVision_Mode : BOOL
VAR_INPUT
	ipChObject : I_CH_OBJECT;
	ipGigEVision_Mode : REFERENCE TO I_GigEVision_Mode;
END_VAR

VAR
	ipTmp : I_GigEVision_Mode;
END_VAR

(* 
   1. Test if the interface exists
   2. Test if the object implements a "Object" interface 
   3. Write reference to interface in parameter
   4. Returne TRUE if succesfull
*)
IF ipChObject <> 0 AND_THEN __QUERYINTERFACE(ipChObject,ipTmp) THEN
	ipGigEVision_Mode := ipTmp;
	ToGigEVision_Mode := TRUE;
END_IF

END_FUNCTION

// FUNCTIONs/Casting/ToVIx2000_Mode
FUNCTION ToVIx2000_Mode : BOOL
VAR_INPUT
	ipChObject : I_CH_OBJECT;
	ipVIx2000_Mode : REFERENCE TO I_VIx2000_Mode;
END_VAR

VAR
	ipTmp : I_VIx2000_Mode;
END_VAR

(* 
   1. Test if the interface exists
   2. Test if the object implements a "Object" interface 
   3. Write reference to interface in parameter
   4. Returne TRUE if succesfull
*)
IF ipChObject <> 0 AND_THEN __QUERYINTERFACE(ipChObject,ipTmp) THEN
	ipVIx2000_Mode := ipTmp;
	ToVIx2000_Mode := TRUE;
END_IF

END_FUNCTION

// FUNCTIONs/Casting/ToIlluminationSingleOutput_Mode
FUNCTION ToIlluminationSingleOutput_Mode : BOOL
VAR_INPUT
	ipChObject : I_CH_OBJECT;
	ipSingleOutput_Mode : REFERENCE TO I_IlluminationSingleOutput_Mode;
END_VAR

VAR
	ipTmp : I_IlluminationSingleOutput_Mode;
END_VAR

(* 
   1. Test if the interface exists
   2. Test if the object implements a "Object" interface 
   3. Write reference to interface in parameter
   4. Returne TRUE if succesfull
*)
IF ipChObject <> 0 AND_THEN __QUERYINTERFACE(ipChObject,ipTmp) THEN
	ipSingleOutput_Mode := ipTmp;
	ToIlluminationSingleOutput_Mode := TRUE;
END_IF

END_FUNCTION

// COMPONENTs/Mode/Separate illumination and camera triggers/FB_VisionMode_Pulse_separate
{attribute 'no_explicit_call' := '[FB_VisionMode_Pulse] Do not call the body - Stick to OOP'}
//Pulse - A trigger activates an image acquisition with simultaneous triggering of the lighting 
FUNCTION_BLOCK FB_VisionMode_Pulse_separate EXTENDS FB_VisionMode_Base IMPLEMENTS I_VisionMode_Pulse_Separate
VAR
	{attribute 'hide'}
	bInitDone : BOOL;
	{attribute 'hide'}
	nLastTriggerTime_Camera : T_DCTIME64;
	{attribute 'hide'}
	nLastTriggerTime_Illumination : T_DCTIME64;
	
	
	(* Supported/requested interfaces. Minimum one must be supported per ImageProvider/CameraController/IlluminationController *)
	(* ImageProvider *)
	ipGigeVision_Mode 		: I_GigEVision_Mode;	
	ipImageFromFile_Mode	: I_ImageFromFile_Mode;	
	
	(* Supported/requested interfaces. Minimum one must be supported per ImageProvider/CameraController/IlluminationController *)
	(* CameraController *)
	ipHwTimestamp_Mode 		: I_HwTimestamp_Mode;
	ipSwTimestamp_Mode		: I_SwTimestamp_Mode;
	ipGigeSoftwaretrigger 	: I_GigeSoftTrigger_Mode;
	
	(* Supported/requested interfaces. Minimum one must be supported per ImageProvider/CameraController/IlluminationController *)
	(* lluminationController 1 *)
	ipVIx2000_Mode_1 		: I_VIx2000_Mode;
	ipSingleOutput_Mode_1 	: I_IlluminationSingleOutput_Mode;
		
	(* Supported/requested interfaces. Minimum one must be supported per ImageProvider/CameraController/IlluminationController *)
	(* lluminationController 2 *)
	ipVIx2000_Mode_2 	: I_VIx2000_Mode;
	ipSingleOutput_Mode_2 	: I_IlluminationSingleOutput_Mode;
	
END_VAR

METHOD Configure : HRESULT
VAR_INPUT
	nOrange 	: UINT(0..511); //0-511
	nGreen 		: UINT(0..511); //0-511
	nBlue 		: UINT(0..511); //0-511
	nInfrared 	: UINT(0..511); //0-511
//	nExposureDelay_100ns : UDINT;	//Camera start at triggertime, illumination starts this time earlier
	nExposure_1us : UDINT;			//Camera 
	nIlluminationDuration_1us: UDINT;
	nIlluminationOverride : USINT(1..100); // 1-100
END_VAR
VAR
	hr : HRESULT;
END_VAR
IF NOT bInitDone THEN
	Configure := E_FAIL;
	RETURN;
END_IF	


(* CameraController *)
(* Decide here how the hardware is to be controlled based on the interface that was found *)
IF ipHwTimestamp_Mode <> 0 THEN
//	ipHwTimestamp_Mode.TriggerDelay_1ns := nExposureDelay_100ns; zzz clean up
	ipHwTimestamp_Mode.Duration_1us := nExposure_1us;// + TO_UDINT(nExposureDelay_100ns/10); //exposure + warm up time
END_IF

IF ipSwTimestamp_Mode <> 0 THEN
//	ipSwTimestamp_Mode.TriggerDelay_1ns := nExposureDelay_100ns;
END_IF

IF ipGigeSoftwaretrigger <> 0 THEN
	ipGigeSoftwaretrigger.GigeCamera := ipGigeVision_Mode;
//	ipGigeSoftwaretrigger.TriggerDelay_1ns := nExposureDelay_100ns;
END_IF
(* -------------------------------------------------------------------------------------------------------- *)


(* ImageProvider *)
(* Decide here how the hardware is to be controlled based on the interface that was found *)
IF ipGigeVision_Mode <> 0 THEN
	ipGigeVision_Mode.Exposure_1us := nExposure_1us;
END_IF
(* -------------------------------------------------------------------------------------------------------- *)




(* lluminationController1 *)
(* Decide here how the hardware is to be controlled based on the interface that was found *)
IF ipVIx2000_Mode_1 <> 0 THEN
	hr := GetMostSignificant(hr, ipVIx2000_Mode_1.Configure(
															nOrange		:= (nOrange*nIlluminationOverride/100), 
															nGreen		:= (nGreen*nIlluminationOverride/100), 
															nBlue		:= (nBlue*nIlluminationOverride/100), 
															nInfrared	:= (nInfrared*nIlluminationOverride/100), 
															nDuration_1us:= nIlluminationDuration_1us));
END_IF
(* -------------------------------------------------------------------------------------------------------- *)




(* lluminationController2 *)
(* Decide here how the hardware is to be controlled based on the interface that was found *)
IF ipVIx2000_Mode_2 <> 0 THEN
	hr := GetMostSignificant(hr, ipVIx2000_Mode_2.Configure(
															nOrange		:= (nOrange*nIlluminationOverride/100), 
															nGreen		:= (nGreen*nIlluminationOverride/100), 
															nBlue		:= (nBlue*nIlluminationOverride/100), 
															nInfrared	:= (nInfrared*nIlluminationOverride/100), 
															nDuration_1us:= nIlluminationDuration_1us));
END_IF
(* -------------------------------------------------------------------------------------------------------- *)



Configure := hr;
END_METHOD

METHOD Initialize : HRESULT
VAR 
	bSupportedCameraController, bSupportedlluminationController1, bSupportedlluminationController2, bSupportedlImageProvider : BOOL;
END_VAR

(* CameraController *)
bSupportedCameraController := 	ToHwTimestamp_Mode(ipCameraTriggerController, ipHwTimestamp_Mode)
							OR 	ToSwTimestamp_Mode(ipCameraTriggerController, ipSwTimestamp_Mode)
							OR 	(ToImageFromFile_Mode(ipImageProvider, ipImageFromFile_Mode) AND ipCameraTriggerController=0)	//No Cameracontrolle is allowed if ImageFromFile				
							OR (ToGigeSoftTrigger_Mode(ipCameraTriggerController, ipGigeSoftwaretrigger) AND ToGigEVision_Mode(ipImageProvider, ipGigeVision_Mode));//GigE Softtrigger requires a GigE ImageProvider
							// OR ...

							
(* ImageProvider *)
bSupportedlImageProvider := ToGigEVision_Mode(ipImageProvider, ipGigeVision_Mode)	
						 OR ToImageFromFile_Mode(ipImageProvider, ipImageFromFile_Mode); 
							// OR ...

							
(* lluminationController1 *)
bSupportedlluminationController1 := 	ToVIx2000_Mode(ipIlluminationController1, ipVIx2000_Mode_1)
									OR 	ToIlluminationSingleOutput_Mode(ipIlluminationController1, ipSingleOutput_Mode_1)
									OR 	(ipIlluminationController1 = 0); //Ilumination1+2 is optional -> Empty or valide
									// OR ...

									
(* lluminationController2 *)
bSupportedlluminationController2 := 	ToVIx2000_Mode(ipIlluminationController2, ipVIx2000_Mode_2)
									OR 	ToIlluminationSingleOutput_Mode(ipIlluminationController2, ipSingleOutput_Mode_2)
									OR 	(ipIlluminationController2 = 0); //Ilumination1+2 is optional -> Empty or valide
									// OR ...

									

bInitDone := bSupportedCameraController AND bSupportedlImageProvider AND bSupportedlluminationController1 AND bSupportedlluminationController2;


IF bInitDone THEN 
	Initialize := S_OK;
ELSE
	Initialize := E_FAIL;
END_IF
END_METHOD

{attribute 'monitoring' := 'call'}
PROPERTY LastTriggerTime_Camera : T_DCTIME64
GET
LastTriggerTime_Camera := nLastTriggerTime_Camera;
END_GET
END_PROPERTY

{attribute 'monitoring' := 'call'}
PROPERTY LastTriggerTime_Illumination : T_DCTIME64
GET
LastTriggerTime_Illumination := nLastTriggerTime_Illumination;
END_GET
END_PROPERTY

{attribute 'monitoring' := 'call'}
// Name or description of this mode
PROPERTY Name : STRING
GET
Name := 'Acquisition with separate triggering of the lighting';
END_GET
END_PROPERTY

METHOD TriggerAtDcTime_Camera : HRESULT
VAR_INPUT
	//The data type T_DCTIME64 represents the distributed clock system time (abbreviated as DC time) as a linear 64-bit integer value. 
	//The time is expressed in nanoseconds since 1/1/2000 UTC. The smallest unit is a nanosecond.
	//F_GetCurDcTickTime64()
	nDCTimeStamp	: T_DCTIME64;
END_VAR
VAR
	hr : HRESULT;
END_VAR
IF NOT bInitDone THEN
	TriggerAtDcTime_Camera := E_FAIL;
	RETURN;
END_IF	

(* Check if the trigger is minimum 3 EtherCat cycles in future *)
IF NOT (nDCTimeStamp >= THIS^.NextPossibleTriggerTime) THEN
	TriggerAtDcTime_Camera := E_FAIL;
	RETURN;
END_IF


(* CameraController *)
(* Decide here how the hardware is to be controlled based on the interface that was found *)
IF ipHwTimestamp_Mode <> 0 THEN
	hr := GetMostSignificant(hr, ipHwTimestamp_Mode.Trigger(nDCTimeStamp));
END_IF
IF ipSwTimestamp_Mode <> 0 THEN
	hr := GetMostSignificant(hr, ipSwTimestamp_Mode.Trigger(nDCTimeStamp));
END_IF
IF ipGigeSoftwaretrigger <> 0 THEN
	hr := GetMostSignificant(hr, ipGigeSoftwaretrigger.Trigger(nDCTimeStamp));
END_IF



(* ImageProvider *)
IF ipImageFromFile_Mode <> 0 THEN
	hr := GetMostSignificant(hr, ipImageFromFile_Mode.Trigger(nDCTimeStamp));
END_IF


IF hr = S_OK THEN
	THIS^.nLastTriggerTime_Camera := nDCTimeStamp;
END_IF

TriggerAtDcTime_Camera := hr;
END_METHOD

METHOD TriggerAtDcTime_Illumination : HRESULT
VAR_INPUT
	//The data type T_DCTIME64 represents the distributed clock system time (abbreviated as DC time) as a linear 64-bit integer value. 
	//The time is expressed in nanoseconds since 1/1/2000 UTC. The smallest unit is a nanosecond.
	//F_GetCurDcTickTime64()
	nDCTimeStamp	: T_DCTIME64;
END_VAR
VAR
	hr : HRESULT;
END_VAR
IF NOT bInitDone THEN
	TriggerAtDcTime_Illumination := E_FAIL;
	RETURN;
END_IF	

(* Check if the trigger is minimum 3 EtherCat cycles in future *)
IF NOT (nDCTimeStamp >= THIS^.NextPossibleTriggerTime) THEN
	TriggerAtDcTime_Illumination := E_FAIL;
	RETURN;
END_IF



(* lluminationController1 *)
(* Decide here how the hardware is to be controlled based on the interface that was found *)
IF ipVIx2000_Mode_1 <> 0 THEN
	hr := GetMostSignificant(hr, ipVIx2000_Mode_1.Trigger(nDCTimeStamp));
END_IF
IF ipSingleOutput_Mode_1 <> 0 THEN
	hr := GetMostSignificant(hr, ipSingleOutput_Mode_1.Trigger(nDCTimeStamp));
END_IF



(* lluminationController2 *)
(* Decide here how the hardware is to be controlled based on the interface that was found *)
IF ipVIx2000_Mode_2 <> 0 THEN
	hr := GetMostSignificant(hr, ipVIx2000_Mode_2.Trigger(nDCTimeStamp));
END_IF
IF ipSingleOutput_Mode_2 <> 0 THEN
	hr := GetMostSignificant(hr, ipSingleOutput_Mode_2.Trigger(nDCTimeStamp));
END_IF

IF hr = S_OK THEN
	THIS^.nLastTriggerTime_Illumination := nDCTimeStamp;
END_IF

TriggerAtDcTime_Illumination := hr;
END_METHOD

METHOD TriggerNow_Camera : HRESULT
(* Trigger the vision system *)
TriggerNow_Camera := THIS^.TriggerAtDcTime_Camera(nDCTimeStamp := THIS^.NextPossibleTriggerTime);
END_METHOD

METHOD TriggerNow_Illumination : HRESULT
(* Trigger the vision system *)
TriggerNow_Illumination := THIS^.TriggerAtDcTime_Illumination(nDCTimeStamp := THIS^.NextPossibleTriggerTime);
END_METHOD

END_FUNCTION_BLOCK

// COMPONENTs/Mode/Separate illumination and camera triggers/I_VisionMode_Pulse_separate
INTERFACE I_VisionMode_Pulse_separate

METHOD Configure : HRESULT
VAR_INPUT
	nOrange 	: UINT(0..511); //0-511
	nGreen 		: UINT(0..511); //0-511
	nBlue 		: UINT(0..511); //0-511
	nInfrared 	: UINT(0..511); //0-511
//	nExposureDelay_100ns : UDINT;	//Camera start delay after illumination start zzz
	nExposure_1us : UDINT;			//Camera 
	nIlluminationDuration_1us: UDINT;
	nIlluminationOverride : USINT(1..100); // 1-100
END_VAR
END_METHOD

{attribute 'monitoring' := 'call'}
PROPERTY LastTriggerTime_Camera : T_DCTIME64
GET
END_GET
END_PROPERTY

{attribute 'monitoring' := 'call'}
PROPERTY LastTriggerTime_Illumination : T_DCTIME64
GET
END_GET
END_PROPERTY

{attribute 'monitoring' := 'call'}
PROPERTY NextPossibleTriggerTime : T_DCTIME64
GET
END_GET
END_PROPERTY

METHOD TriggerAtDcTime_Camera : HRESULT
VAR_INPUT
	//The data type T_DCTIME64 represents the distributed clock system time (abbreviated as DC time) as a linear 64-bit integer value. 
	//The time is expressed in nanoseconds since 1/1/2000 UTC. The smallest unit is a nanosecond.
	//F_GetCurDcTickTime64()
	nDCTimeStamp	: T_DCTIME64;
END_VAR
END_METHOD

METHOD TriggerAtDcTime_Illumination : HRESULT
VAR_INPUT
	//The data type T_DCTIME64 represents the distributed clock system time (abbreviated as DC time) as a linear 64-bit integer value. 
	//The time is expressed in nanoseconds since 1/1/2000 UTC. The smallest unit is a nanosecond.
	//F_GetCurDcTickTime64()
	nDCTimeStamp	: T_DCTIME64;
END_VAR
END_METHOD

METHOD TriggerNow_Camera : HRESULT
END_METHOD

METHOD TriggerNow_Illumination : HRESULT
END_METHOD

END_INTERFACE

// COMPONENTs/VisionSystem/FB_VisionSystem
{attribute 'no_explicit_call' := 'Do not call the body - Stick to OOP'}
FUNCTION_BLOCK FB_VisionSystem EXTENDS FB_CH_Object IMPLEMENTS I_VisionSystem
VAR
	{attribute 'hide'}
	ipImageProvider 			: I_ImageProvider_Base;
	{attribute 'hide'}
	ipCameraTriggerController  	: I_CameraTriggerController_Base;
	{attribute 'hide'}
	ipIlluminationController1 	: I_IlluminationController_Base;
	{attribute 'hide'}
	ipIlluminationController2 	: I_IlluminationController_Base;
	{attribute 'hide'}
	ipActiveVisionMode			: I_VisionMode_Base;
	
	{attribute 'hide'}	
	bInitDone 					: BOOL;
	{attribute 'hide'}
	bMethodeExecuteError		: BOOL;
	{attribute 'hide'}
	nPlcTaskCycleTime 			: UDINT; // In 100ns
END_VAR

{attribute 'monitoring' := 'call'}
PROPERTY ActiveMode : I_VisionMode_StatusOnly
GET
ActiveMode := ipActiveVisionMode;
END_GET
END_PROPERTY

{attribute 'monitoring' := 'call'}
PROPERTY CameraController : I_CameraTriggerController_StatusOnly
GET
CameraController := ipCameraTriggerController;
END_GET
END_PROPERTY

{attribute 'monitoring' := 'call'}
PROPERTY IlluminationController1 : I_IlluminationController_StatusOnly
GET
IlluminationController1 := ipIlluminationController1;
END_GET
END_PROPERTY

{attribute 'monitoring' := 'call'}
PROPERTY IlluminationController2 : I_IlluminationController_StatusOnly
GET
IlluminationController2 := ipIlluminationController2;
END_GET
END_PROPERTY

{attribute 'monitoring' := 'call'}
PROPERTY ImageProvider : I_ImageProvider_StatusOnly
GET
ImageProvider := ipImageProvider;
END_GET
END_PROPERTY

METHOD FB_exit : BOOL
VAR_INPUT
	bInCopyCode : BOOL; // if TRUE, the exit method is called for exiting an instance that is copied afterwards (online change).
END_VAR
VAR
	pUkn : POINTER TO ITcUnknown;
END_VAR
//IF THIS^.iVisionMode <> 0 AND_THEN __QUERYPOINTER(THIS^.iVisionMode, pUkn) THEN
//	THIS^.iVisionMode := 0;
//	FW_SafeRelease(PipUnk := ADR(pUkn));
//END_IF
END_METHOD

{attribute 'monitoring' := 'call'}
// Name or description of the active mode
PROPERTY ActiveModeName : STRING
GET
IF  THIS^.ipActiveVisionMode <> 0 THEN
	ActiveModeName := THIS^.ipActiveVisionMode.Name;
ELSE
	ActiveModeName := 'No mode selected or error during activation';
END_IF
END_GET
END_PROPERTY

METHOD SetMode : HRESULT
VAR_INPUT
	ipAnyMode : I_VisionMode_Base;
END_VAR
VAR 
	hr : HRESULT;
END_VAR
IF ipAnyMode = 0 THEN
	//Error, invalide input
	SetMode := E_FAIL;
	RETURN;
END_IF

//Set new Mode
THIS^.ipActiveVisionMode := ipAnyMode;

//Handover interface to componets
hr := GetMostSignificant(hr, THIS^.ipActiveVisionMode.LinkComponents(
														ipVisionSystem 	:= THIS^,
														ipImageProvider 		:= THIS^.ipImageProvider, 
														ipCameraTriggerController 		:= THIS^.ipCameraTriggerController, 
														ipIlluminationController1 := THIS^.ipIlluminationController1, 
														ipIlluminationController2 := THIS^.ipIlluminationController2));
	
hr := GetMostSignificant(hr, THIS^.ipActiveVisionMode.Initialize());

IF (hr <> S_OK) THEN
	//Reject new mode on error during link or initialize
	THIS^.ipActiveVisionMode := 0;
END_IF

SetMode := hr;
END_METHOD

{attribute 'monitoring' := 'call'}
//Module already has a task - already a trigger active
PROPERTY Busy : BOOL
GET
VAR
	bBusy : BOOL;
END_VAR
IF THIS^.ipImageProvider <> 0 THEN
	bBusy := bBusy OR THIS^.ipImageProvider.Feedback.Busy;
END_IF

IF THIS^.ipCameraTriggerController <> 0 THEN
	bBusy := bBusy OR THIS^.ipCameraTriggerController.Feedback.Busy;
END_IF

IF THIS^.ipIlluminationController1 <> 0 THEN
	bBusy := bBusy OR THIS^.ipIlluminationController1.Busy;
END_IF

IF THIS^.ipIlluminationController2 <> 0 THEN
	bBusy := bBusy OR THIS^.ipIlluminationController2.Busy;
END_IF

Busy := bBusy;
END_GET
END_PROPERTY

{attribute 'monitoring' := 'call'}
PROPERTY Error : BOOL  // Module started successfully and entered aquiring mode
GET
VAR
	bError : BOOL := FALSE;;
END_VAR
IF THIS^.ipImageProvider <> 0 THEN
	bError := bError OR THIS^.ipImageProvider.State = ETcVnCameraState.TCVN_CS_ERROR;
END_IF

IF THIS^.ipCameraTriggerController <> 0 THEN
	bError := bError OR THIS^.ipCameraTriggerController.State = E_StateTerminal.ERROR;
END_IF

IF THIS^.ipIlluminationController1 <> 0 THEN
	bError := bError OR THIS^.ipIlluminationController1.State = E_StateTerminal.ERROR;
END_IF

IF THIS^.ipIlluminationController2 <> 0 THEN
	bError := bError OR THIS^.ipIlluminationController2.State = E_StateTerminal.ERROR;
END_IF


Error := bError;
END_GET
END_PROPERTY

METHOD FB_init : BOOL
VAR_INPUT
	bInitRetains : BOOL; // if TRUE, the retain variables are initialized (warm start / cold start)
	bInCopyCode : BOOL;  // if TRUE, the instance afterwards gets moved into the copy code (online change)
	
	ipImageProvider 			: I_ImageProvider_Base;	
	ipCameraTriggerController  	: I_CameraTriggerController_Base;
	ipIlluminationController1 	: I_IlluminationController_Base;
	ipIlluminationController2 	: I_IlluminationController_Base;

END_VAR
VAR_INST
	{attribute 'hide'}
	bFBInitCalledOnce : BOOL; //Do the following code once during start up and not during onlinechange
END_VAR
//Do the following code once during start up and not during onlinechange
IF NOT bFBInitCalledOnce THEN 
	
	THIS^.ipImageProvider 				:= ipImageProvider;
	THIS^.ipCameraTriggerController 	:= ipCameraTriggerController;
	THIS^.ipIlluminationController1 	:= ipIlluminationController1;
	THIS^.ipIlluminationController2 	:= ipIlluminationController2;

END_IF

bFBInitCalledOnce := TRUE;
END_METHOD

METHOD Initialize : HRESULT
VAR
	hr : HRESULT;
END_VAR
VAR_INST
	bParentSet : BOOL;
END_VAR
THIS^.nPlcTaskCycleTime(*100ns*) := TwinCAT_SystemInfoVarList._TaskInfo[THIS^.TaskIndex].CycleTime;

//(* Validate all inputs *)
//IF (iImageProvider = 0 OR iCameraController = 0 )THEN
//	Initialize := E_FAIL;
//	RETURN;
//END_IF

IF NOT bParentSet THEN
	bParentSet := TRUE;
	
	IF ipCameraTriggerController <> 0 THEN
		THIS^.ipCameraTriggerController.SetParent(THIS^);
	END_IF		
	
	IF ipImageProvider <> 0 THEN
		THIS^.ipImageProvider.SetParent(THIS^);
	END_IF		
	
	IF ipIlluminationController1 <> 0 THEN
		THIS^.ipIlluminationController1.SetParent(THIS^);
	END_IF	
	
	IF ipIlluminationController2 <> 0 THEN
		THIS^.ipIlluminationController2.SetParent(THIS^);
	END_IF
END_IF

hr := SUPER^.Initialize();

IF ipImageProvider <> 0 THEN
	hr := GetMostSignificant(hr, THIS^.ipImageProvider.Initialize());
END_IF	
IF ipCameraTriggerController <> 0 THEN
	hr := GetMostSignificant(hr, THIS^.ipCameraTriggerController.Initialize());
END_IF	
IF ipIlluminationController1 <> 0 THEN
	hr := GetMostSignificant(hr, THIS^.ipIlluminationController1.Initialize());
END_IF	
IF ipIlluminationController2 <> 0 THEN
	hr := GetMostSignificant(hr, THIS^.ipIlluminationController2.Initialize());
END_IF	


IF CheckOk(hr) THEN
	bInitDone := TRUE;
END_IF


bMethodeExecuteError := bMethodeExecuteError OR FAILED(hr);


Initialize := hr;
END_METHOD

{attribute 'monitoring':='call'}
PROPERTY Initialized : BOOL
GET
Initialized := THIS^.bInitDone;
END_GET
END_PROPERTY

{attribute 'monitoring' := 'call'}
PROPERTY OID : OTCID
GET
IF THIS^.ipImageProvider <> 0 THEN
	OID := THIS^.ipImageProvider.OID;
ELSE
	OID := SUPER^.OID;
END_IF
END_GET
END_PROPERTY

{attribute 'monitoring' := 'call'}
PROPERTY Operational : BOOL  // Module started successfully and entered aquiring mode
GET
VAR
	bReady : BOOL := TRUE;;
END_VAR
IF THIS^.ipImageProvider <> 0 THEN
	bReady := bReady AND THIS^.ipImageProvider.Operational;
END_IF

IF THIS^.ipCameraTriggerController <> 0 THEN
	bReady := bReady AND THIS^.ipCameraTriggerController.Operational;
END_IF

IF THIS^.ipIlluminationController1 <> 0 THEN
	bReady := bReady AND THIS^.ipIlluminationController1.Operational;
END_IF

IF THIS^.ipIlluminationController2 <> 0 THEN
	bReady := bReady AND THIS^.ipIlluminationController2.Operational;
END_IF

Operational := bReady AND NOT THIS^.Error;
END_GET
END_PROPERTY

METHOD Reset : HRESULT
VAR
	hr : HRESULT;
END_VAR
IF NOT bInitDone THEN
	Reset := E_FAIL;
	RETURN;
END_IF

IF ipImageProvider <> 0 THEN
	hr := GetMostSignificant(hr, THIS^.ipImageProvider.Reset());
END_IF

IF ipCameraTriggerController <> 0 THEN
	hr := GetMostSignificant(hr, THIS^.ipCameraTriggerController.Reset());
END_IF

IF ipIlluminationController1 <> 0 THEN
	hr := GetMostSignificant(hr, THIS^.ipIlluminationController1.Reset());
END_IF
	
IF ipIlluminationController2 <> 0 THEN
	hr := GetMostSignificant(hr, THIS^.ipIlluminationController2.Reset());
END_IF	


bMethodeExecuteError := FALSE;
bMethodeExecuteError := bMethodeExecuteError OR FAILED(hr);

Reset := hr;
END_METHOD

{attribute 'monitoring' := 'call'}
PROPERTY TaskCycleTimeNs : UDINT // Set task cycle time in multiples of 100 ns
GET
TaskCycleTimeNs := THIS^.nPlcTaskCycleTime * 100;
END_GET
END_PROPERTY

METHOD TryGetImage : HRESULT
VAR_INPUT
	stImageWithInfo	: REFERENCE TO ST_ImageWithInfo;
END_VAR
IF THIS^.ipImageProvider <> 0 THEN
	TryGetImage := THIS^.ipImageProvider.TryGetImage(stImageWithInfo);
ELSE
	TryGetImage := E_FAIL;
END_IF
END_METHOD

METHOD Update : HRESULT
VAR
	hr : HRESULT;
END_VAR
IF NOT bInitDone THEN
	Update := E_FAIL;
	RETURN;
END_IF

hr := SUPER^.Update();

IF ipCameraTriggerController <> 0 THEN
	hr := GetMostSignificant(hr, THIS^.ipCameraTriggerController.Update());
END_IF

IF ipImageProvider <> 0 THEN
	hr := GetMostSignificant(hr, THIS^.ipImageProvider.Update());
END_IF

IF ipIlluminationController1 <> 0 THEN
	hr := GetMostSignificant(hr, THIS^.ipIlluminationController1.Update());
END_IF
	
IF ipIlluminationController2 <> 0 THEN
	hr := GetMostSignificant(hr, THIS^.ipIlluminationController2.Update());
END_IF	

IF THIS^.ipActiveVisionMode <> 0 THEN
	hr := GetMostSignificant(hr, THIS^.ipActiveVisionMode.Update());
END_IF


bMethodeExecuteError := bMethodeExecuteError OR FAILED(hr);

Update := hr;
END_METHOD

END_FUNCTION_BLOCK

// COMPONENTs/VnRegister-Access/FB_VnRegister_REAL
{attribute 'no_explicit_call' := 'Do not call the body - Stick to OOP'}
FUNCTION_BLOCK FB_VnRegister_REAL EXTENDS FB_VnRegister_Base
VAR
	{attribute 'hide'}
	fValue : REAL;
	
	{attribute 'hide'}	
	fbVnReadRegister_REAL : FB_VN_ReadRegister_REAL;
	{attribute 'hide'}	
	fbVnWriteRegister_REAL : FB_VN_WriteRegister_REAL;
END_VAR

METHOD FB_init : BOOL
VAR_INPUT
	bInitRetains : BOOL; // if TRUE, the retain variables are initialized (warm start / cold start)
	bInCopyCode : BOOL;  // if TRUE, the instance afterwards gets moved into the copy code (online change)
	
	ipCameraConnection : I_GigEVision_Register_Connection;
	nAddress : GVCP_REGISTER_ADDRESS;
    nEndian  : UINT;
END_VAR
VAR_INST
	{attribute 'hide'}
	bFBInitCalledOnce : BOOL; //Do the following code once during start up and not during onlinechange
END_VAR
//Do the following code once during start up and not during onlinechange
IF NOT bFBInitCalledOnce THEN 
	nCtsVnRegisterObject := nCtsVnRegisterObject +1;
	

	THIS^.nEndian 		:= nEndian;
	
	//Copy ObjectId from Camera to this fbVnReadRegister.
	MEMCPY(destAddr := ADR(fbVnReadRegister_REAL.oidITcVnGevImageProvider), srcAddr:=ADR(SUPER^.OidCamera), n:= SIZEOF(SUPER^.OidCamera));
	MEMCPY(destAddr := ADR(fbVnWriteRegister_REAL.oidITcVnGevImageProvider), srcAddr:=ADR(SUPER^.OidCamera), n:= SIZEOF(SUPER^.OidCamera));

	//Force to do an init after set OID
	fbVnReadRegister_REAL.FB_init(FALSE,FALSE);	
	fbVnWriteRegister_REAL.FB_init(FALSE,FALSE);
END_IF

bFBInitCalledOnce := TRUE;
END_METHOD

METHOD Update : HRESULT
SUPER^.Update();


fbVnReadRegister_REAL(
	nAddress:= SUPER^.nAddress, 
	nEndian:= SUPER^.nEndian, 
	bRead:= SUPER^.bExecuteRead, 
	fValue=> fValue, 
	bBusy=> SUPER^.bReadBusy, 
	bError=> SUPER^.bReadError
	);
IF fbRTrigReadDone.Q AND THIS^.bWriteDone THEN
	fValue := fbVnReadRegister_REAL.fValue;
END_IF
	
fbVnWriteRegister_REAL(
	nAddress:= SUPER^.nAddress, 
	fValue:= fValue,  
	nEndian:= SUPER^.nEndian,   
	bWrite:= SUPER^.bExecuteWrite, 
	bBusy=> SUPER^.bWriteBusy, 
	bError=> SUPER^.bWriteError,
	);
END_METHOD

{attribute 'monitoring':='call'}
PROPERTY Value : REAL
GET
Value := fValue;
END_GET
SET
fValue := Value;

//Trigger a new write cycle
THIS^.bWriteDone 	:= FALSE;
END_SET
END_PROPERTY

END_FUNCTION_BLOCK

// COMPONENTs/VnRegister-Access/FB_VnRegister_ULINT
{attribute 'no_explicit_call' := 'Do not call the body - Stick to OOP'}
FUNCTION_BLOCK FB_VnRegister_ULINT EXTENDS FB_VnRegister_Base
VAR
	{attribute 'hide'}
	nValue : ULINT;
	
	{attribute 'hide'}	
	fbVnReadRegister_ULINT : FB_VN_ReadRegister_ULINT;
	{attribute 'hide'}	
	fbVnWriteRegister_ULINT : FB_VN_WriteRegister_ULINT;
END_VAR

METHOD FB_init : BOOL
VAR_INPUT
	bInitRetains : BOOL; // if TRUE, the retain variables are initialized (warm start / cold start)
	bInCopyCode : BOOL;  // if TRUE, the instance afterwards gets moved into the copy code (online change)
	
	ipCameraConnection : I_GigEVision_Register_Connection;
	nAddress : GVCP_REGISTER_ADDRESS;
    nEndian  : UINT;
END_VAR
VAR_INST
	{attribute 'hide'}
	bFBInitCalledOnce : BOOL; //Do the following code once during start up and not during onlinechange
END_VAR
//Do the following code once during start up and not during onlinechange
IF NOT bFBInitCalledOnce THEN 
	nCtsVnRegisterObject := nCtsVnRegisterObject +1;
	

	THIS^.nEndian 		:= nEndian;
	
	//Copy ObjectId from Camera to this fbVnReadRegister.
	MEMCPY(destAddr := ADR(fbVnReadRegister_ULINT.oidITcVnGevImageProvider), srcAddr:=ADR(SUPER^.OidCamera), n:= SIZEOF(SUPER^.OidCamera));
	MEMCPY(destAddr := ADR(fbVnWriteRegister_ULINT.oidITcVnGevImageProvider), srcAddr:=ADR(SUPER^.OidCamera), n:= SIZEOF(SUPER^.OidCamera));

	//Force to do an init after set OID
	fbVnReadRegister_ULINT.FB_init(FALSE,FALSE);	
	fbVnWriteRegister_ULINT.FB_init(FALSE,FALSE);
END_IF

bFBInitCalledOnce := TRUE;
END_METHOD

METHOD Update : HRESULT
SUPER^.Update();


fbVnReadRegister_ULINT(
	nAddress:= SUPER^.nAddress, 
	nEndian:= SUPER^.nEndian, 
	bRead:= SUPER^.bExecuteRead, 
	nValue=> nValue, 
	bBusy=> SUPER^.bReadBusy, 
	bError=> SUPER^.bReadError
	);
IF fbRTrigReadDone.Q AND THIS^.bWriteDone THEN
	nValue := fbVnReadRegister_ULINT.nValue;
END_IF
	
fbVnWriteRegister_ULINT(
	nAddress:= SUPER^.nAddress, 
	nValue:= nValue,  
	nEndian:= SUPER^.nEndian,   
	bWrite:= SUPER^.bExecuteWrite, 
	bBusy=> SUPER^.bWriteBusy, 
	bError=> SUPER^.bWriteError,
	);
END_METHOD

{attribute 'monitoring':='call'}
PROPERTY Value : ULINT
GET
Value := nValue;
END_GET
SET
nValue := Value;

//Trigger a new write cycle
THIS^.bWriteDone 	:= FALSE;
END_SET
END_PROPERTY

END_FUNCTION_BLOCK

// FUNCTIONs/Casting/ToCameraController
FUNCTION ToCameraController : BOOL
VAR_INPUT
	ipChObject : I_CH_OBJECT;
	ipTriggerSource : REFERENCE TO I_CameraTriggerController_Base;
END_VAR

VAR
	ipTmp : I_CameraTriggerController_Base;
END_VAR

(* 
   1. Test if the interface exists
   2. Test if the object implements a "Object" interface 
   3. Write reference to interface in parameter
   4. Returne TRUE if succesfull
*)
IF ipChObject <> 0 AND_THEN __QUERYINTERFACE(ipChObject,ipTmp) THEN
	ipTriggerSource := ipTmp;
	ToCameraController := TRUE;
END_IF

END_FUNCTION

// FUNCTIONs/Casting/ToImageProvider
FUNCTION ToImageProvider : BOOL
VAR_INPUT
	ipChObject : I_CH_OBJECT;
	ipImageProvider : REFERENCE TO I_ImageProvider_Base;
END_VAR

VAR
	ipTmp : I_ImageProvider_Base;
END_VAR

(* 
   1. Test if the interface exists
   2. Test if the object implements a "Object" interface 
   3. Write reference to interface in parameter
   4. Returne TRUE if succesfull
*)
IF ipChObject <> 0 AND_THEN __QUERYINTERFACE(ipChObject,ipTmp) THEN
	ipImageProvider := ipTmp;
	ToImageProvider := TRUE;
END_IF

END_FUNCTION

// FUNCTIONs/Casting/TolluminationController
FUNCTION TolluminationController : BOOL
VAR_INPUT
	ipChObject : I_CH_OBJECT;
	ipLigthSource : REFERENCE TO I_IlluminationController_Base;
END_VAR

VAR
	ipTmp : I_IlluminationController_Base;
END_VAR

(* 
   1. Test if the interface exists
   2. Test if the object implements a "Object" interface 
   3. Write reference to interface in parameter
   4. Returne TRUE if succesfull
*)
IF ipChObject <> 0 AND_THEN __QUERYINTERFACE(ipChObject,ipTmp) THEN
	ipLigthSource := ipTmp;
	TolluminationController := TRUE;
END_IF

END_FUNCTION

// FUNCTIONs/Casting/ToVisionMode_Pulse_combined
FUNCTION ToVisionMode_Pulse_combined : BOOL
VAR_INPUT
	ipChObject : I_CH_OBJECT;
	ipVisionMode_Pulse : REFERENCE TO I_VisionMode_Pulse_combined;
END_VAR

VAR
	ipTmp : I_VisionMode_Pulse_combined;
END_VAR

(* 
   1. Test if the interface exists
   2. Test if the object implements a "Object" interface 
   3. Write reference to interface in parameter
   4. Returne TRUE if succesfull
*)
IF ipChObject <> 0 AND_THEN __QUERYINTERFACE(ipChObject,ipTmp) THEN
	ipVisionMode_Pulse := ipTmp;
	ToVisionMode_Pulse_combined := TRUE;
END_IF

END_FUNCTION

// FUNCTIONs/Casting/ToVisionMode_Pulse_separate
FUNCTION ToVisionMode_Pulse_separate : BOOL
VAR_INPUT
	ipChObject : I_CH_OBJECT;
	ipVisionMode_Pulse : REFERENCE TO I_VisionMode_Pulse_separate;
END_VAR

VAR
	ipTmp : I_VisionMode_Pulse_separate;
END_VAR

(* 
   1. Test if the interface exists
   2. Test if the object implements a "Object" interface 
   3. Write reference to interface in parameter
   4. Returne TRUE if succesfull
*)
IF ipChObject <> 0 AND_THEN __QUERYINTERFACE(ipChObject,ipTmp) THEN
	ipVisionMode_Pulse := ipTmp;
	ToVisionMode_Pulse_separate := TRUE;
END_IF

END_FUNCTION

// FUNCTIONs/Color/F_ColorEnumToVector4
FUNCTION F_ColorEnumToVector4 : TcVnVector4_LREAL
VAR_INPUT
	eColor : E_Color_ARGB;
END_VAR
VAR
	nValue : DWORD; //0-255
END_VAR

//R
nValue := SHR((eColor AND 16#00FF0000), 4*4);
F_ColorEnumToVector4[0] := DWORD_TO_LREAL(nValue);

//G
nValue := SHR((eColor AND 16#0000FF00), 2*4);
F_ColorEnumToVector4[1] := DWORD_TO_LREAL(nValue);

//B
nValue := SHR((eColor AND 16#000000FF), 0*4);
F_ColorEnumToVector4[2] := DWORD_TO_LREAL(nValue);

//A
nValue := SHR((eColor AND 16#FF000000), 6*4);
F_ColorEnumToVector4[3] := DWORD_TO_LREAL(nValue);

END_FUNCTION

// FUNCTIONs/Sharpness/F_VND_Sharpness_SumModifiedLaplace_ULINT
FUNCTION F_VND_Sharpness_SumModifiedLaplace_ULINT : HRESULT
VAR_INPUT
	ipImg			: REFERENCE TO ITcVnImage;	
	nKernelSize		: USINT; //3 or 5
	hrPrev			: HRESULT;
END_VAR
VAR_OUTPUT
	nSharpness		: ULINT:=0;
END_VAR
VAR
	ppData			: POINTER TO REAL;
	ipTmp			: ITcVnImage;
	ipImgData		: ITcVnData;
	nDataSize		: ULINT;
	nJ				: ULINT;
END_VAR

//Bad error has occurred in the previous processing chain
IF FAILED(hrPrev) THEN
	F_VND_Sharpness_SumModifiedLaplace_ULINT := hrPrev;
	RETURN;
END_IF

//Invalide input
IF ipImg = 0 THEN
    F_VND_Sharpness_SumModifiedLaplace_ULINT := Tc2_System.E_HRESULTAdsErr.INVALIDPARM;
    RETURN;
END_IF

hrPrev := F_VN_LaplacianFilterExp(
	ipSrcImage:=ipImg, 
	ipDestImage:=ipTmp, 
	eDestDepth:=ETcVnElementType.TCVN_ET_REAL, 
	nKernelSize:=nKernelSize, 
	fScale:=1, 
	fDelta:=0, 
	eBorderType:=ETcVnBorderInterpolationMethod.TCVN_BIM_DEFAULT, 
	hrPrev:=hrPrev);

ipTmp.GetImageData(
	pipImageData:=ADR(ipImgData));

ipImgData.GetDataPointer(
	ppData:=ADR(ppData));

ipImgData.GetSize(
	nSize:=nDataSize);

FOR nJ:=0 TO nDataSize/4-1 DO
	nSharpness := nSharpness + TO_ULINT(ABS(ppData[nJ]));
END_FOR

ipImgData.ReleaseDataPointer(ppData:=ADR(ppData));
FW_SafeRelease(pipUnk:=ADR(ipImgData));
FW_SafeRelease(pipUnk:=ADR(ipTmp));

F_VND_Sharpness_SumModifiedLaplace_ULINT := hrPrev;

END_FUNCTION
